INTERFACE I_LoggedEventsSort

METHOD Sort : HRESULT
VAR_IN_OUT
	aLoggedEvents : T_LoggedEvents;
END_VAR
END_METHOD

END_INTERFACE

(* stored: Version 1.1.0.1, ProductVersion 3.1.4024.12
   Itf I_LoggedEventsSort: Id {87711ce4-569b-402b-a71b-c008fb0eaeaf}
   Method Sort: Id {b4fe590f-a95d-4ee0-b977-a958029d9023} *)
